(* Logix 5000 project; controller Conveyer_vfd_Ethernetip_simulation vendor 1 type 14 code 196 rev 36.11; software revision 36.00 *)

TASK MainTask (continuous, watchdog 500 ms) : MainProgram

MODULES
   Local : vendor 1 type 14 code 196 (5069 0, rev 36.11)
END_MODULES

TYPE UDT_VFD_INTERFACE :   // Simulated Ethernet/Ip vfd interface including command, reference, status, and feedback signals
STRUCT
   LogicCommand : DINT;   // command word sent to vfd
   Reference : INT;   // speed reference (0.01 Hz)
   LogicStatus : DINT;   // drive status word
   Feedback : INT;   // speed feedback (0.01 Hz)
   FaultCode : INT;   // simulated drive fault code
   Ready : BOOL;   // drive ready status
   active : BOOL;   // drive running status
   foward : BOOL;   // foward direction status
   Faulted : BOOL;   // drive fault status
   AtSpeed : BOOL;   // drive at speed status
END_STRUCT
END_TYPE

VAR_GLOBAL   (* controller tags *)
   Auto_Runreq : BOOL;
   Cmd_Reset : BOOL;
   Cmd_Run : BOOL;
   Cmd_Speed_Hz : REAL;
   Cmd_Stop : BOOL;
   Conv_AtSpeed : BOOL;
   Conv_LoadPct : REAL;
   Conv_ProductPresent : BOOL;
   Conv_RunFb : BOOL;
   Conv_SpeedCmd_Hz : REAL;
   Conv_SpeedFb_Hz : REAL;
   Conv_SpeedPct : REAL;
   MachineState : DINT;   // Conveyor machine operating state
   Manual_RunCmd : BOOL;
   Manual_Speed_Hz : REAL;
   Max_Speed_Hz : REAL;   // 60.0
   Min_Speed_Hz : REAL;   // 0.0
   Mode_Auto : BOOL;
   Mode_Manual : BOOL;
   PB_ESTOP_OK : BOOL;
   PB_GUARDDOOR_OK : BOOL;
   PB_RESETFAULT : BOOL;
   PB_START : BOOL;
   PB_STOP : BOOL;
   Permissive_Runok : BOOL;
   Ramp_Accel_HzPerSec : REAL;   // 5.0
   Ramp_Decel_HzPerSec : REAL;   // 7.0
   Sim_CommFault : BOOL;
   Sim_DriverFault : BOOL;
   Sim_Overload : BOOL;
   System_Fault : BOOL;
   Task_DT : REAL;   // 0.02
   temp_Reference : REAL;
   VFD_Conveyor : UDT_VFD_INTERFACE;
   VFD_FaultCode : INT;
   VFD_Feedback : INT;
   VFD_LogicCommand : DINT;
   VFD_LogisticStatus : DINT;
   VFD_Reference : INT;
END_VAR

PROGRAM MainProgram   (* main routine MainRoutine *)
VAR
   Base_LoadPct : REAL := 20.0;   // 20.0
   Drive_RunReq : BOOL;
   HighSpeed_LoadPct : REAL;   // 10.0
   OL_DelayTimer : TIMER := (PRE := 3000);
   OL_ThresholdPct : REAL := 95.0;   // 95.0
   Product_LoadPct : REAL := 15.0;   // 15.0
   Ref_Hz : REAL;
   SpeedError : DINT;
   SpeedStep : REAL;
   Temp_SpeedError : REAL;
END_VAR

ROUTINE MainRoutine   (* ladder *)
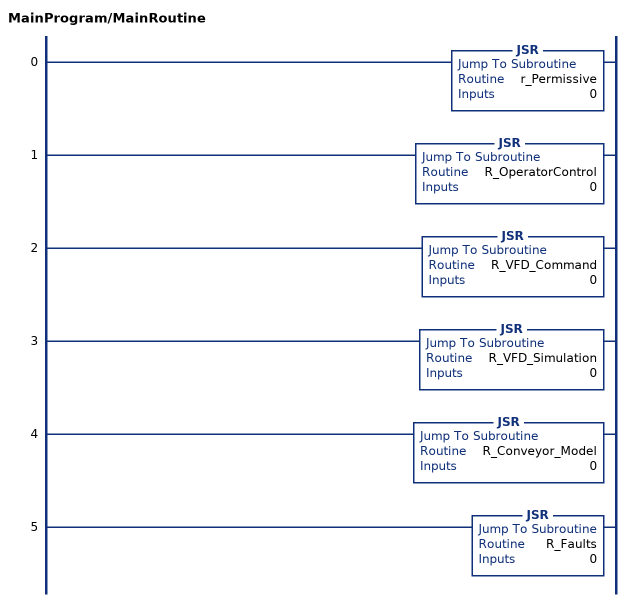
   0: JSR(r_Permissive,0);
   1: JSR(R_OperatorControl,0);
   2: JSR(R_VFD_Command,0);
   3: JSR(R_VFD_Simulation,0);
   4: JSR(R_Conveyor_Model,0);
   5: JSR(R_Faults,0);
END_ROUTINE

ROUTINE R_Conveyor_Model   (* ladder *)
// This routine simulates conveyor behavior. It calculates conveyor load based on speed and product presence and generates overload conditions when load exceeds safe limits
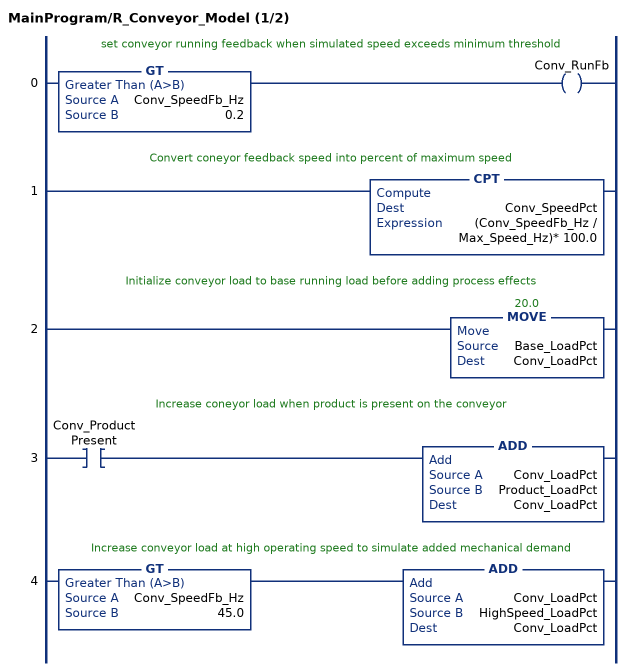
   // set conveyor running feedback when simulated speed exceeds minimum threshold
   0: GT(Conv_SpeedFb_Hz,0.2)OTE(Conv_RunFb);
   // Convert coneyor feedback speed into percent of maximum speed
   1: CPT(Conv_SpeedPct,(Conv_SpeedFb_Hz / Max_Speed_Hz)* 100.0);
   // Initialize conveyor load to base running load before adding process effects
   2: MOVE(Base_LoadPct,Conv_LoadPct);
   // Increase coneyor load when product is present on the conveyor
   3: XIC(Conv_ProductPresent)ADD(Conv_LoadPct,Product_LoadPct,Conv_LoadPct);
   // Increase conveyor load at high operating speed to simulate added mechanical demand
   4: GT(Conv_SpeedFb_Hz,45.0)ADD(Conv_LoadPct,HighSpeed_LoadPct,Conv_LoadPct);
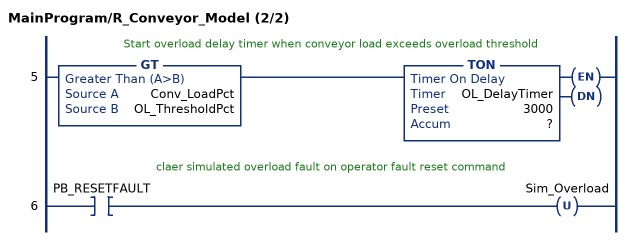
   // Start overload delay timer when conveyor load exceeds overload threshold
   5: GT(Conv_LoadPct,OL_ThresholdPct)TON(OL_DelayTimer,?,?);
   // claer simulated overload fault on operator fault reset command
   6: XIC(PB_RESETFAULT)OTU(Sim_Overload);
END_ROUTINE

ROUTINE R_Faults   (* ladder *)
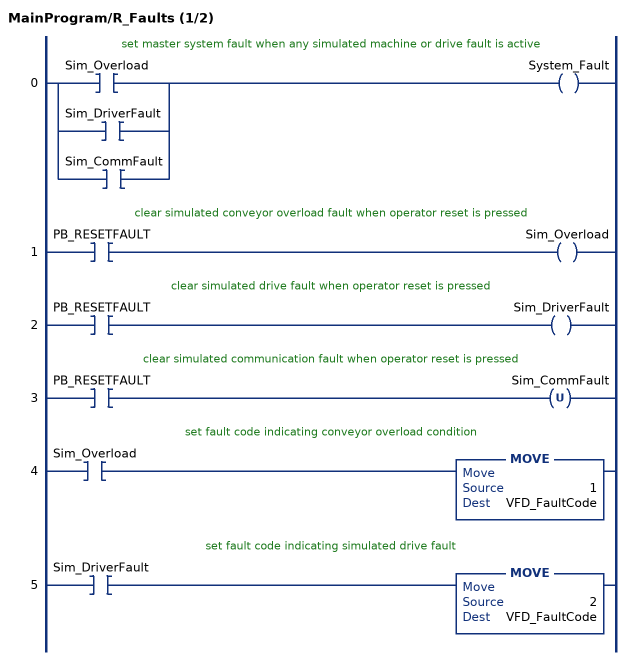
   // set master system fault when any simulated machine or drive fault is active
   0: [XIC(Sim_Overload) ,[XIC(Sim_DriverFault) ,XIC(Sim_CommFault) ] ]OTE(System_Fault);
   // clear simulated conveyor overload fault when operator reset is pressed
   1: XIC(PB_RESETFAULT)OTE(Sim_Overload);
   // clear simulated drive fault when operator reset is pressed
   2: XIC(PB_RESETFAULT)OTE(Sim_DriverFault);
   // clear simulated communication fault when operator reset is pressed
   3: XIC(PB_RESETFAULT)OTU(Sim_CommFault);
   // set fault code indicating conveyor overload condition
   4: XIC(Sim_Overload)MOVE(1,VFD_FaultCode);
   // set fault code indicating simulated drive fault
   5: XIC(Sim_DriverFault)MOVE(2,VFD_FaultCode);
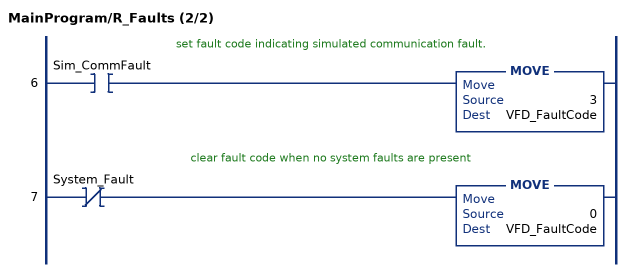
   // set fault code indicating simulated communication fault.
   6: XIC(Sim_CommFault)MOVE(3,VFD_FaultCode);
   // clear fault code when no system faults are present
   7: XIO(System_Fault)MOVE(0,VFD_FaultCode);
END_ROUTINE

ROUTINE R_OperatorControl   (* ladder *)
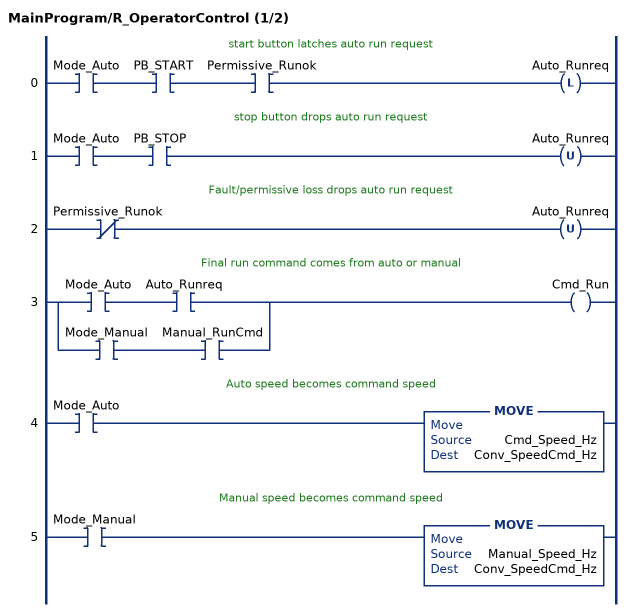
   // start button latches auto run request
   0: XIC(Mode_Auto)XIC(PB_START)XIC(Permissive_Runok)OTL(Auto_Runreq);
   // stop button drops auto run request
   1: XIC(Mode_Auto)XIC(PB_STOP)OTU(Auto_Runreq);
   // Fault/permissive loss drops auto run request
   2: XIO(Permissive_Runok)OTU(Auto_Runreq);
   // Final run command comes from auto or manual
   3: [XIC(Mode_Auto) XIC(Auto_Runreq) ,XIC(Mode_Manual) XIC(Manual_RunCmd) ]OTE(Cmd_Run);
   // Auto speed becomes command speed
   4: XIC(Mode_Auto)MOVE(Cmd_Speed_Hz,Conv_SpeedCmd_Hz);
   // Manual speed becomes command speed
   5: XIC(Mode_Manual)MOVE(Manual_Speed_Hz,Conv_SpeedCmd_Hz);
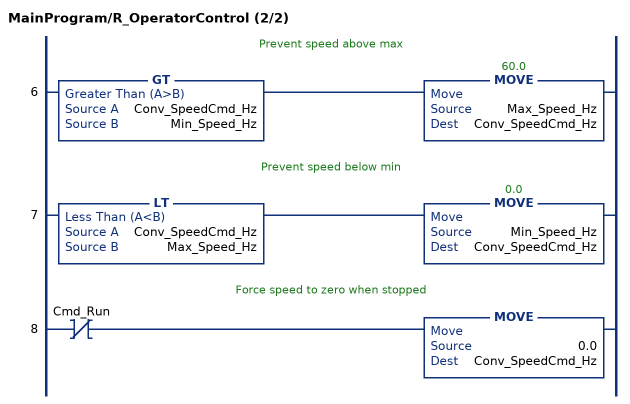
   // Prevent speed above max
   6: GT(Conv_SpeedCmd_Hz,Min_Speed_Hz)MOVE(Max_Speed_Hz,Conv_SpeedCmd_Hz);
   // Prevent speed below min
   7: LT(Conv_SpeedCmd_Hz,Max_Speed_Hz)MOVE(Min_Speed_Hz,Conv_SpeedCmd_Hz);
   // Force speed to zero when stopped
   8: XIO(Cmd_Run)MOVE(0.0,Conv_SpeedCmd_Hz);
END_ROUTINE

ROUTINE r_Permissive   (* ladder *)
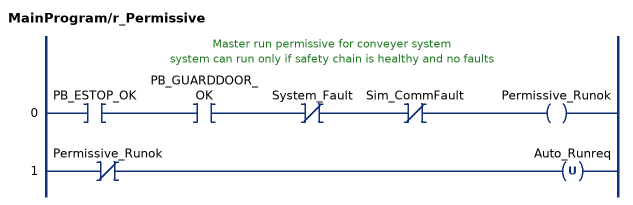
   // Master run permissive for conveyer system
   // system can run only if safety chain is healthy and no faults
   0: XIC(PB_ESTOP_OK)XIC(PB_GUARDDOOR_OK)XIO(System_Fault)XIO(Sim_CommFault)OTE(Permissive_Runok);
   1: XIO(Permissive_Runok)OTU(Auto_Runreq);
END_ROUTINE

ROUTINE R_StateMachine   (* ladder *)
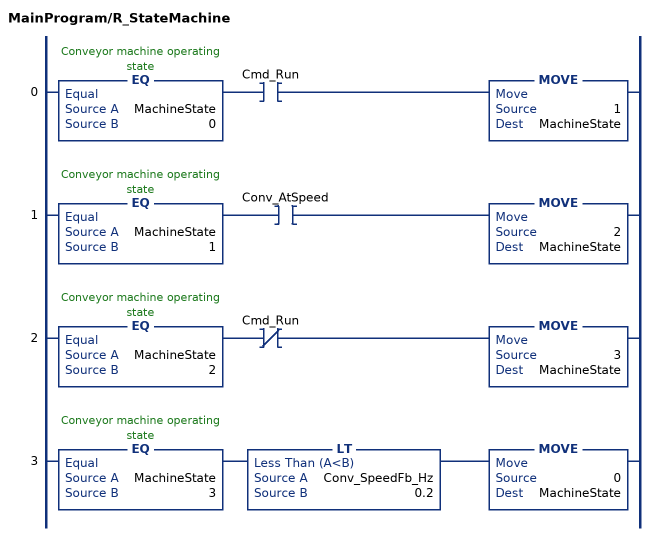
   0: EQ(MachineState,0)XIC(Cmd_Run)MOVE(1,MachineState);
   1: EQ(MachineState,1)XIC(Conv_AtSpeed)MOVE(2,MachineState);
   2: EQ(MachineState,2)XIO(Cmd_Run)MOVE(3,MachineState);
   3: EQ(MachineState,3)LT(Conv_SpeedFb_Hz,0.2)MOVE(0,MachineState);
END_ROUTINE

ROUTINE R_VFD_Command   (* ladder *)
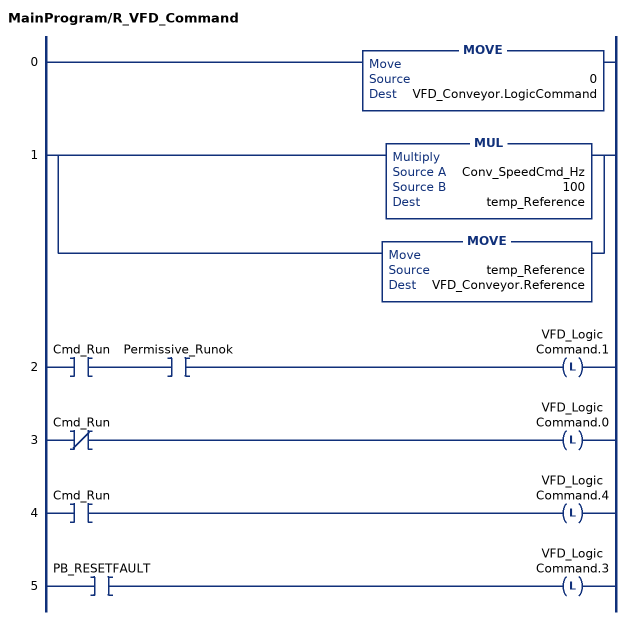
   0: MOVE(0,VFD_Conveyor.LogicCommand);
   1: [MUL(Conv_SpeedCmd_Hz,100,temp_Reference) ,MOVE(temp_Reference,VFD_Conveyor.Reference) ];
   2: XIC(Cmd_Run)XIC(Permissive_Runok)OTL(VFD_LogicCommand.1);
   3: XIO(Cmd_Run)OTL(VFD_LogicCommand.0);
   4: XIC(Cmd_Run)OTL(VFD_LogicCommand.4);
   5: XIC(PB_RESETFAULT)OTL(VFD_LogicCommand.3);
END_ROUTINE

ROUTINE R_VFD_Simulation   (* ladder *)
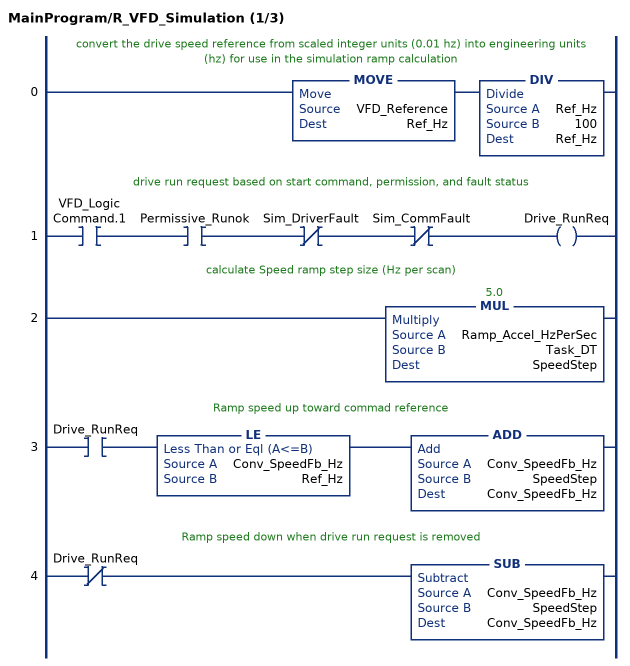
   // convert the drive speed reference from scaled integer units (0.01 hz) into engineering units (hz) for use in the simulation ramp calculation
   0: MOVE(VFD_Reference,Ref_Hz)DIV(Ref_Hz,100,Ref_Hz);
   // drive run request based on start command, permission, and fault status
   1: XIC(VFD_LogicCommand.1)XIC(Permissive_Runok)XIO(Sim_DriverFault)XIO(Sim_CommFault)OTE(Drive_RunReq);
   // calculate Speed ramp step size (Hz per scan)
   2: MUL(Ramp_Accel_HzPerSec,Task_DT,SpeedStep);
   // Ramp speed up toward commad reference
   3: XIC(Drive_RunReq)LE(Conv_SpeedFb_Hz,Ref_Hz)ADD(Conv_SpeedFb_Hz,SpeedStep,Conv_SpeedFb_Hz);
   // Ramp speed down when drive run request is removed
   4: XIO(Drive_RunReq)SUB(Conv_SpeedFb_Hz,SpeedStep,Conv_SpeedFb_Hz);
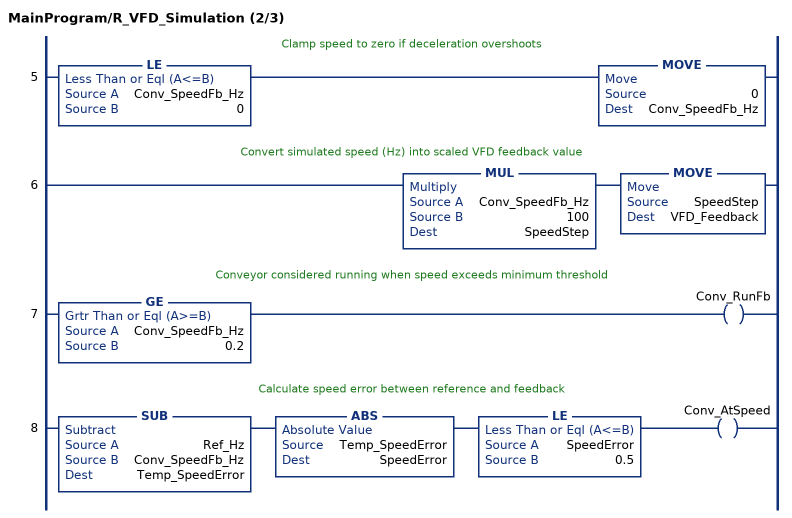
   // Clamp speed to zero if deceleration overshoots
   5: LE(Conv_SpeedFb_Hz,0)MOVE(0,Conv_SpeedFb_Hz);
   // Convert simulated speed (Hz) into scaled VFD feedback value
   6: MUL(Conv_SpeedFb_Hz,100,SpeedStep)MOVE(SpeedStep,VFD_Feedback);
   // Conveyor considered running when speed exceeds minimum threshold
   7: GE(Conv_SpeedFb_Hz,0.2)OTE(Conv_RunFb);
   // Calculate speed error between reference and feedback
   8: SUB(Ref_Hz,Conv_SpeedFb_Hz,Temp_SpeedError)ABS(Temp_SpeedError,SpeedError)LE(SpeedError,0.5)OTE(Conv_AtSpeed);
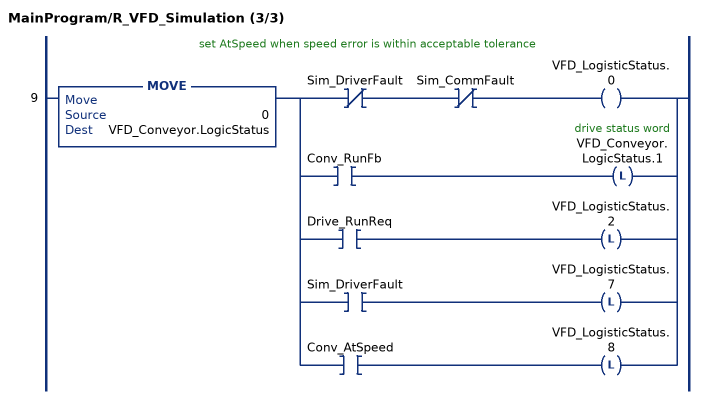
   // set AtSpeed when speed error is within acceptable tolerance
   9: MOVE(0,VFD_Conveyor.LogicStatus)[XIO(Sim_DriverFault) XIO(Sim_CommFault) OTE(VFD_LogisticStatus.0) ,[XIC(Conv_RunFb) OTL(VFD_Conveyor.LogicStatus.1) ,[XIC(Drive_RunReq) OTL(VFD_LogisticStatus.2) ,[XIC(Sim_DriverFault) OTL(VFD_LogisticStatus.7) ,XIC(Conv_AtSpeed) OTL(VFD_LogisticStatus.8) ] ] ] ];
END_ROUTINE
END_PROGRAM
